// TwinCAT 3 PLC project TwinCAT_OpenFramework_Tasks
// Title: TwinCAT Open Framework Tasks
// Company: Oleksandr Tiutyk FOP
// Author: Oleksandr Tiutyk
// ProjectVersion: 1.0.13.0
// Description: TwinCAT.OpenFramework abstractions to run simple tasks
// ProgramVersion: 3.1.4026.28
// libraries:
//   [TwinCAT Open Framework Collections], * (Oleksandr Tiutyk FOP)
//   [TwinCAT Open Framework Core], * (Oleksandr Tiutyk FOP)
// project tree:
//   Internal/ CurrentNamespace.TcPOU, NamespaceExtractor.TcPOU
//   TaskQueue/ StandardTaskQueue.TcPOU (not stored), TaskQueue.TcPOU
//   Task/Enums/ TASK_PROCESSING_STATE.TcDUT (not stored), TASK_RUNNING_SUBSTATE.TcDUT, TASK_STATE.TcDUT (not stored), TASK_STOP_REASON.TcDUT (not stored)
//   Task/ ITask.TcIO, Task.TcPOU
//   Task/SubObjects/ TaskRunningSubstate.TcPOU (not stored), TaskState.TcPOU, TaskStopReason.TcPOU (not stored)
//   Version/ Global_Version.TcGVL
// (motion and I/O tree: see PLC project twincat_openframework_core)
// real-time tasks:
//   TASK PlcTask: cycle T#10ms, priority 20, ADS port 350
//   TASK TestTask: cycle T#10ms, priority 1, ADS port 351
//   TASK RunnerTestTask: cycle T#10ms, priority 2, ADS port 354
//   TASK HowToTask: cycle T#10ms, priority 22, ADS port 353
// variable links:

// ---- Task/Enums/TASK_RUNNING_SUBSTATE.TcDUT
(*
SPDX-FileCopyrightText: © 2026 Oleksandr Tiutyk <trofimich@gmail.com>
SPDX-License-Identifier: MIT
License: https://opensource.org/license/mit
*)

(*!
<summary>Identifies the active phase of a running task.</summary>
<description>
Acquisition, processing, stopping and release are diagnostic substates, not independent scheduling tasks.
Interpret them only while TASK_STATE is RUNNING.
</description>
*)
{attribute 'qualified_only'}
{attribute 'strict'}
{attribute 'to_string'}
TYPE TASK_RUNNING_SUBSTATE :
(
	//! <summary>Acquire the resource before ordinary work.</summary>
	RESOURCE_ACQUIRING := 0,
	//! <summary>Advance ordinary work unless cancellation is pending.</summary>
	PROCESSING,
	//! <summary>Advance the terminal resource-release attempt.</summary>
	RESOURCE_RELEASING,
	//! <summary>Finish active work for any stop reason before resource release.</summary>
	STOPPING
);
END_TYPE

// ---- Version/Global_Version.TcGVL
{attribute 'TcGenerated'}
{attribute 'no-analysis'}
{attribute 'linkalways'}
// This function has been automatically generated from the project information.
VAR_GLOBAL CONSTANT
	{attribute 'const_non_replaced'}
	stLibVersion_TwinCAT_Open_Framework_Tasks : ST_LibVersion := (iMajor := 1, iMinor := 0, iBuild := 13, iRevision := 0, nFlags := 0, sVersion := '1.0.13.0');
END_VAR

// ---- Task/ITask.TcIO
(*
SPDX-FileCopyrightText: © 2026 Oleksandr Tiutyk <trofimich@gmail.com>
SPDX-License-Identifier: MIT
License: https://opensource.org/license/mit
*)

(*!
<summary>Defines a reusable cooperative operation with optional resource acquisition and release.</summary>
<description>
One owner drives inherited Execute cyclically while RUNNING, including after an accepted Cancel, until
STOPPED. Avoid concurrent or recursive Execute on the same task. State, RunningSubstate and stop reasons are
borrowed live views for observation only; keep the task alive and do not modify referenced data. Copy result
values and messages before Reset or reuse. Boolean control results do not establish a general no-throw
guarantee for arbitrary implementations or diagnostic failures.
</description>
*)
INTERFACE ITask EXTENDS TOF_Core.IExecutable, TOF_Core.INamed

(*!
<summary>Requests cancellation before resource release begins.</summary>
<description>
Accepted only in RUNNING with no pending cancellation and before resource release. TRUE means accepted, not
completed; continue Execute until STOPPED. Accepted cancellation enters STOPPING, including from a previous
work result in that phase, and sets EXTERNAL_CANCEL. Repeated, releasing or non-running requests return FALSE
with refuseReason.
</description>
<param name="refuseReason">Reason for refusal; meaningful on FALSE.</param>
*)
METHOD Cancel : BOOL
VAR_OUTPUT
	refuseReason : TOF_Core.ERROR_MESSAGE;
END_VAR
END_METHOD

(*!
<summary>Provides the final lifecycle result for a stopped task.</summary>
<description>
Meaningful as a final result only in STOPPED. Release exceptions produce FAILURE without an automatic release
retry; STOPPED does not prove physical resource release. Best-effort errors handled inside the manager do not
by themselves change this result. Reset clears the message and restores the default reason. The view is
borrowed and read-only.
</description>
*)
{attribute 'monitoring' := 'call'}

PROPERTY FINAL FinalStopReason : REFERENCE TO TaskStopReason
GET
END_GET
END_PROPERTY

(*!
<summary>Provides the reason that initiated stopping.</summary>
<description>
Completion, internal abort, external cancellation or failure is preserved with its message during release; a
release exception affects FinalStopReason instead. The initial WORK_DONE value does not indicate completion.
Reset restores defaults. This is a borrowed read-only live view.
</description>
*)
{attribute 'monitoring' := 'call'}

PROPERTY FINAL OriginalStopReason : REFERENCE TO TaskStopReason
GET
END_GET
END_PROPERTY

(*!
<summary>Prepares a stopped task for reuse.</summary>
<description>
READY returns TRUE without callbacks or reinitialization. RUNNING refuses reset; cancel and keep calling
Execute until STOPPED first. In STOPPED, successful reset restores default stop reasons and clears their
messages. A refused reset does not guarantee rollback of callback effects.
</description>
<param name="refuseReason">Reason for refusal; meaningful on FALSE.</param>
*)
METHOD Reset : BOOL
VAR_OUTPUT
	refuseReason : TOF_Core.ERROR_MESSAGE;
END_VAR
END_METHOD

(*!
<summary>Provides the borrowed manager used by the task, or zero for none.</summary>
<description>
Keep the manager alive and stable throughout the run. The task issues StartAcquire or StartRelease once per
phase and advances Execute; external callers must not drive those operations concurrently. Pending acquisition
and active work must finish according to the concrete manager and task contracts before release.
ResourceManager and ResourceAcquired getters have no side effects and must not throw.
</description>
*)
{attribute 'monitoring' := 'call'}

PROPERTY ResourceManager : TOF_Core.IResourceManager
GET
END_GET
END_PROPERTY

(*!
<summary>Provides a live diagnostic view of the running phase.</summary>
<description>
Meaningful only while State.Running is TRUE. Observe acquisition, processing, stopping or release without
driving the resource manager directly. The view is borrowed and read-only.
</description>
*)
{attribute 'monitoring' := 'call'}

PROPERTY FINAL RunningSubstate : REFERENCE TO TaskRunningSubstate
GET
END_GET
END_PROPERTY

(*!
<summary>Starts a READY task's lifecycle.</summary>
<description>
TRUE means RUNNING, not completed. Continue Execute for work and cleanup. Ineligible state or refused
preparation returns FALSE with refuseReason. Refusal does not guarantee rollback of preparation already
performed.
</description>
<param name="refuseReason">Reason for refusal; meaningful on FALSE.</param>
*)
METHOD Start : BOOL
VAR_OUTPUT
	refuseReason : TOF_Core.ERROR_MESSAGE;
END_VAR
END_METHOD

(*!
<summary>Provides a live view of the task lifecycle.</summary>
<description>
READY precedes start, RUNNING includes acquisition, work, stopping and release, and STOPPED marks termination.
Assess the completed result through FinalStopReason. StateChanged is cleared at the start of Execute and set
on a lifecycle transition; its lifetime follows method calls, not necessarily one PLC cycle. The view is
borrowed and read-only.
</description>
*)
{attribute 'monitoring' := 'call'}

PROPERTY FINAL State : REFERENCE TO TaskState
GET
END_GET
END_PROPERTY

END_INTERFACE

// ---- Internal/CurrentNamespace.TcPOU
(*
SPDX-FileCopyrightText: © 2026 Oleksandr Tiutyk <trofimich@gmail.com>
SPDX-License-Identifier: MIT
License: https://opensource.org/license/mit
*)

(*!
<summary>Exposes this library's compiler-initialized namespace.</summary>
<description>
Internal metadata provider; no cyclic body call is needed. The returned namespace is borrowed read-only
storage.
</description>
*)

{attribute 'no_explicit_call' := 'do not call this POU directly'}
PROGRAM INTERNAL CurrentNamespace
VAR
	{attribute 'hide'} 
	_NamespaceExtractor : NamespaceExtractor;
END_VAR

(*!
<summary>Borrows the compiler-initialized library namespace.</summary>
<description>
Do not modify the referenced storage. Reading does not allocate or transfer ownership.
</description>
*)
{attribute 'monitoring' := 'call'}
PROPERTY Name : REFERENCE TO STRING
GET
Name REF= _NamespaceExtractor.CurrentNamespace;
END_GET
END_PROPERTY

END_PROGRAM

// ---- Internal/NamespaceExtractor.TcPOU
(*
SPDX-FileCopyrightText: © 2026 Oleksandr Tiutyk <trofimich@gmail.com>
SPDX-License-Identifier: MIT
License: https://opensource.org/license/mit
*)

(*!
<summary>Captures the current library namespace through init_namespace.</summary>
<description>
The compiler initializes CurrentNamespace. The empty body requires no execution; consumers treat the output as
read-only metadata.
</description>
*)

FUNCTION_BLOCK INTERNAL NamespaceExtractor
VAR_OUTPUT
	//! <summary>Compiler-supplied library namespace; read-only to consumers.</summary>
	{attribute 'init_namespace'} 
	CurrentNamespace : STRING;	
END_VAR

END_FUNCTION_BLOCK

// ---- TaskQueue/TaskQueue.TcPOU
(*
SPDX-FileCopyrightText: © 2026 Oleksandr Tiutyk <trofimich@gmail.com>
SPDX-License-Identifier: MIT
License: https://opensource.org/license/mit
*)

(*!
<summary>Executes borrowed child tasks sequentially in FIFO order.</summary>
<description>
One owner drives the queue and the lifecycles of its queued children. Children must be live, READY when
enqueued and unique in this queue; callers must not independently drive them while queued. Only one child is
active at a time. The dynamic list owns its storage but not child objects. Successful children are removed;
unsuccessful current and waiting entries remain until cleared or reset. Empty queues keep running unless
StopWhenNoPendingTasks is TRUE. All stop reasons advance the current child's cleanup without starting waiting
children. The base Task records a processing exception and enters STOPPING; OnStopping requests child
cancellation and waits for completion before parent release. An accepted external Cancel during that wait
retains the base Task cancellation result; the first failure is submitted to the log. No cleanup timeout is
imposed. Descendants overriding queue hooks must preserve the inherited queue operations.
</description>
*)

{attribute 'no_explicit_call' := 'do not call this function block directly'}
FUNCTION_BLOCK ABSTRACT TaskQueue EXTENDS Task
VAR
	{attribute 'hide'} 
	_SubTasks : TOF_Collections.List<0>(0);
	
	{attribute 'hide'} 
	_CurrentTask : ITask;
	
	{attribute 'hide'} 
	_StopWhenNoPendingTasks : BOOL;
END_VAR

(*!
<summary>Removes waiting entries without resetting or deleting child objects.</summary>
<description>
While RUNNING with a current task, retains that first entry and removes the rest. Otherwise clears all entries
and the current reference. Does not request cancellation. A stopped unsuccessful current task is removed when
clearing outside RUNNING.
</description>
*)
METHOD FINAL ClearWaitingTasks
VAR
	i : DINT;
END_VAR
IF NOT State.Running OR_ELSE _CurrentTask = 0 THEN
	_SubTasks.Clear();
	_CurrentTask := 0;
ELSE	
	FOR i := _SubTasks.Length - 1 TO 1 BY -1 DO
		_SubTasks.RemoveAt(index := i);
	END_FOR
END_IF
END_METHOD

(*!
<summary>Appends a prepared borrowed task to the FIFO.</summary>
<description>
Null raises ArgumentNotSpecifiedException. READY and uniqueness are caller preconditions, not checked here.
Keep the child alive and do not start, execute, cancel or reset it independently while queued. Removal
transfers no ownership and does not reset or delete it. No queue-state guard is applied; Reset from STOPPED
clears entries, so prepare the queue before filling it for reuse. Storage growth can raise terminal allocation
failure.
</description>
<param name="task">Live READY child whose lifecycle is delegated to the queue until removal.</param>
*)
METHOD PROTECTED FINAL EnqueueTask
VAR_INPUT
	task : ITask;
END_VAR
VAR
	
	taskAsGeneric : TOF_Core.GENERIC_VALUE;
END_VAR
IF task = 0 THEN
	TOF_Core.Exceptions.ThrowArgumentNotSpecified(
		sourceNamespaceName := NamespaceName,
		sourceClassName := ClassName,
		sourcePOUName := __POUNAME(),
		sourcePosition := __POSITION(),
		argumentName := 'task'
	);
END_IF

taskAsGeneric := TOF_Core.GenericValueFactory.FromParts(
		genericTypeClass := TOF_Core.GENERIC_TYPE_CLASS.OBJECT,
		address := task.SelfAddress,
		size := task.SelfSize,
		memoryManagementBehavior := TOF_Core.GENERIC_MEMORY_MANAGEMENT_BEHAVIOR.STORE_ORIGINAL_REFERENCE_AND_NOT_OWNS_MEMORY
	);

_SubTasks.AppendGeneric(value := taskAsGeneric);
END_METHOD

(*!
<summary>Resolves one stored entry to its task interface.</summary>
<description>
Requires a valid zero-based index and a live borrowed child. List access rejects an invalid index; failure to
query ITask raises StandardException. Does not clone or transfer ownership.
</description>
<param name="index">Index within the queue's current list.</param>
*)
METHOD PRIVATE getTaskByIndex : ITask
VAR_INPUT
	index : DINT;
END_VAR
VAR
	taskInterface : TOF_Core.IObject;
	
END_VAR
taskInterface := _SubTasks.Get(index := index).AsIObject();

IF NOT __QUERYINTERFACE(taskInterface, getTaskByIndex) THEN
	TOF_Core.Exceptions.ThrowStandard(
		sourceNamespaceName := NamespaceName,
		sourceClassName := ClassName,
		sourcePOUName := __POUNAME(),
		sourcePosition := __POSITION(),
		message := "Can't convert task from _Tasks collection to ITask type"
	);
END_IF
END_METHOD

(*!
<summary>Cancels and advances the current child before any parent termination.</summary>
<description>
Called by the common STOPPING phase after any result or exception. Never starts waiting children. Requests
Cancel while the child is RUNNING, then advances it once. A Cancel exception is contained so Execute still
gets a chance to progress; readiness remains FALSE for that call. Execute exceptions reach the base stopping
handler, which retains the original result and retries. Refusal of Cancel does not imply completion. No child
is removed or reset here. Additional descendant cleanup must combine readiness with this result.
</description>
<param name="readyToRelease">TRUE when no child is RUNNING and this stopping step completed normally.</param>
*)
METHOD PROTECTED OnStopping
VAR_OUTPUT
	readyToRelease : BOOL;
END_VAR
VAR
	cancelCallFailed : BOOL;
END_VAR
IF _CurrentTask <> 0 AND_THEN _CurrentTask.State.Running THEN
	__TRY
		_CurrentTask.Cancel();
	__CATCH
		// Advance the child even if its cancellation request was interrupted.
		cancelCallFailed := TRUE;
	__ENDTRY

	_CurrentTask.Execute();
END_IF

readyToRelease := NOT cancelCallFailed
	AND_THEN (_CurrentTask = 0 OR_ELSE NOT _CurrentTask.State.Running);
END_METHOD

(*!
<summary>Forwards an accepted queue cancellation to its running child.</summary>
<description>
Called once by the task's Cancel path. Does not wait or inspect the child's refusal message; a child already
stopping can refuse another cancellation request. OnStopping advances completion. Preserve forwarding when
overriding this hook.
</description>
*)
METHOD PROTECTED OnCancelRequest
IF _CurrentTask <> 0 AND_THEN _CurrentTask.State.Running THEN
	_CurrentTask.Cancel();
END_IF
END_METHOD

(*!
<summary>Clears a stopped queue for reuse.</summary>
<description>
Releases list storage and drops current and waiting references without resetting or deleting children. Their
owner prepares them before re-enqueueing. Base Reset clears stop diagnostics. READY Reset does not invoke this
hook; use ClearWaitingTasks to empty a READY queue. Descendants must preserve this step.
</description>
*)
METHOD PROTECTED OnReset
_SubTasks.Clear();
_CurrentTask := 0;
END_METHOD

(*!
<summary>Starts or advances at most one current child per processing call.</summary>
<description>
An existing current child receives one Execute. Otherwise the first waiting child is selected and started;
newly started work is advanced by a later call. Start refusal or an unexpected READY current yields ERROR. A
successful stopped child is removed; other results are mapped from FinalStopReason and its message. An empty
queue yields DONE only when StopWhenNoPendingTasks is TRUE. Removing the last successful child leaves BUSY
until the next call. Exceptions propagate to the base Task failure handler, which records and logs diagnostics
and enters STOPPING. OnStopping waits for child cleanup before parent release.
</description>
<param name="processingState">Queue progress; defaults to BUSY while waiting or advancing a child.</param>
<param name="stopReasonMessage">Receives child refusal or unsuccessful completion diagnostics.</param>
*)
METHOD PROTECTED OnRunning
VAR_OUTPUT
	processingState : TASK_PROCESSING_STATE;
END_VAR
VAR_IN_OUT
	stopReasonMessage : TOF_Core.ERROR_MESSAGE;
END_VAR
IF _CurrentTask <> 0 THEN
	_CurrentTask.Execute();
ELSIF _SubTasks.Length > TOF_Core.SignedInt32.ZERO THEN
	_CurrentTask := getTaskByIndex(index := 0);

	IF NOT _CurrentTask.Start(refuseReason => stopReasonMessage) THEN
		processingState := TASK_PROCESSING_STATE.ERROR;
		RETURN;
	END_IF
ELSIF _StopWhenNoPendingTasks THEN
	processingState := TASK_PROCESSING_STATE.DONE;
END_IF

IF _CurrentTask <> 0 THEN
	CASE _CurrentTask.State.Value OF
		TASK_STATE.READY:
			processingState := TASK_PROCESSING_STATE.ERROR;
			stopReasonMessage := "Current task returned to READY before completion";

		TASK_STATE.STOPPED:
			IF _CurrentTask.FinalStopReason.WorkDone THEN
				removeCurrentTask();
			ELSE
				processingState := GetProcessingStateByStopReason(taskStopReason := _CurrentTask.FinalStopReason.Value);
				stopReasonMessage := _CurrentTask.FinalStopReason.Message;
			END_IF
	END_CASE
END_IF
END_METHOD

(*!
<summary>Reports the number of entries still retained by the queue.</summary>
<description>
Includes the current task and waiting children, including a failed or cancelled current retained after
stopping. Zero does not by itself mean the queue has reached STOPPED.
</description>
*)
{attribute 'monitoring' := 'call'}
PROPERTY FINAL PendingTaskCount : DINT
GET
PendingTaskCount := _SubTasks.Length;
END_GET
END_PROPERTY

(*!
<summary>Removes the first queue entry and clears the current reference.</summary>
<description>
Used after successful child completion. Compacts remaining list entries without resetting or deleting the
child; the caller retains its object and may inspect its stopped result. Does not start the next child.
</description>
*)
METHOD PRIVATE removeCurrentTask
IF _SubTasks.Length > 0 THEN
	_SubTasks.RemoveAt(index := 0);
END_IF

_CurrentTask := 0;
END_METHOD

(*!
<summary>Controls whether an empty running queue completes.</summary>
<description>
Defaults to FALSE, allowing Execute to wait for later enqueueing. TRUE makes OnRunning report DONE when it
finds no current or waiting child. May be changed between owner calls; setting it does not itself execute or
stop the queue.
</description>
*)
{attribute 'monitoring' := 'call'}
PROPERTY FINAL StopWhenNoPendingTasks : BOOL
GET
StopWhenNoPendingTasks := _StopWhenNoPendingTasks;
END_GET
SET
_StopWhenNoPendingTasks := StopWhenNoPendingTasks;
END_SET
END_PROPERTY

END_FUNCTION_BLOCK

// ---- Task/Task.TcPOU
(*
SPDX-FileCopyrightText: © 2026 Oleksandr Tiutyk <trofimich@gmail.com>
SPDX-License-Identifier: MIT
License: https://opensource.org/license/mit
*)

(*!
<summary>Runs a reusable cooperative operation through acquisition, processing, stopping and release.</summary>
<description>
One owner drives the task through Start, cyclic Execute and Reset; no worker thread or PLC scheduler task is
created. Keep callbacks short and avoid concurrent or recursive Execute. The resource manager is borrowed and
must remain live and stable during a run. All stop reasons wait through OnStopping before release. Normal work
completion advances stopping in the same Execute, without waiting or repeating work. No callback may
recursively drive this task, except Reset in OnAfterStop. Ordinary work and resource exceptions are converted
into stop diagnostics where handled. If obtaining their messages fails, phase-specific fallback text preserves
the intended failure transition; preparation and reset use the same fallback policy for refusal. The first
stopping exception is submitted to the log; later stopping exceptions retry without repeated log attempts.
This is not a universal no-throw boundary. The caller still provides exception cleanup and terminal
allocation-failure checks at its PLC task boundary. DiagnosticLogger optionally selects an independent
diagnostic channel; zero preserves LogManager routing. Configure it before Start and keep it stable until
STOPPED, including Reset diagnostics, with no concurrent access.
</description>
*)

{attribute 'no_explicit_call' := 'do not call this function block directly'}
FUNCTION_BLOCK ABSTRACT Task EXTENDS TOF_Core.Object IMPLEMENTS ITask
VAR
	{attribute 'hide'} 
	_Name : WSTRING;

	//! <summary>Optional borrowed destination for this task's internal diagnostics.</summary>
	_DiagnosticLogger : TOF_Core.ILogger;
	
	{attribute 'hide'} 
	_State : TASK_STATE;	
	{attribute 'hide'} 
	_StateChanged : BOOL;	
	{attribute 'hide'} 
	_RunningSubstate : TASK_RUNNING_SUBSTATE;
	{attribute 'hide'} 
	_ResourceOperationStarted : BOOL;
	//! <summary>Tracks whether a stopping exception has been submitted to the log in this run.</summary>
	{attribute 'hide'}
	_StoppingExceptionReportAttempted : BOOL;

	{attribute 'hide'} 
	_OriginalStopReason : TASK_STOP_REASON;
	{attribute 'hide'} 
	_TemporaryErrorMessage : TOF_Core.ERROR_MESSAGE;	
	{attribute 'hide'} 
	_OriginalStopReasonMessage : TOF_Core.ERROR_MESSAGE;
	{attribute 'hide'} 
	_OriginalStopReasonObject : TaskStopReason(_OriginalStopReason, _OriginalStopReasonMessage);
	
	{attribute 'hide'} 
	_FinalStopReason : TASK_STOP_REASON;	
	{attribute 'hide'} 
	_FinalStopReasonMessage : TOF_Core.ERROR_MESSAGE;
	{attribute 'hide'} 
	_FinalStopReasonObject : TaskStopReason(_FinalStopReason, _FinalStopReasonMessage);
	
	{attribute 'hide'} 
	_StateObject : TaskState(_State, _StateChanged);
	{attribute 'hide'} 
	_RunningSubstateObject : TaskRunningSubstate(_RunningSubstate);
END_VAR

(*!
<summary>Requests cooperative cancellation of a running task.</summary>
<description>
Accepted only while RUNNING, with no pending cancellation and before RESOURCE_RELEASING. Records
EXTERNAL_CANCEL as the original reason and enters STOPPING before invoking OnCancelRequest once. A first
Cancel during STOPPING replaces the original result with EXTERNAL_CANCEL. TRUE means accepted, not completed;
continue Execute until STOPPED. Repeated or ineligible requests return FALSE with refuseReason. Callback
exceptions are logged without withdrawing the request.
</description>
<param name="refuseReason">Reason for refusal; meaningful when the method returns FALSE.</param>
*)
METHOD FINAL Cancel : BOOL
VAR_OUTPUT
	refuseReason : TOF_Core.ERROR_MESSAGE;
END_VAR
IF _State <> TASK_STATE.RUNNING THEN
	refuseReason := TOF_Core.WideStrings.Concat255(
		"Expected state is '",
		TO_WSTRING(TASK_STATE.RUNNING),
		"' but current state is '",
		TO_WSTRING(_State),
		"'"
	);
	RETURN;
END_IF

IF _OriginalStopReason = TASK_STOP_REASON.EXTERNAL_CANCEL
	OR_ELSE _RunningSubstate = TASK_RUNNING_SUBSTATE.RESOURCE_RELEASING
THEN
	refuseReason := "Cancellation already requested or resource release has begun";
	RETURN;
END_IF

_OriginalStopReason := TASK_STOP_REASON.EXTERNAL_CANCEL;
_OriginalStopReasonMessage := "Cancelled by external logic";

setRunningSubstate(runningSubState := TASK_RUNNING_SUBSTATE.STOPPING);

safeCallOnCancelRequest();

Cancel := TRUE;
END_METHOD

(*!
<summary>Advances the running task and clears its transition indicator.</summary>
<description>
Clears State.StateChanged on every call, including READY and STOPPED calls. While RUNNING, advances
acquisition, work or release without a blocking wait. A normal terminal work result also advances stopping
once in the same call. A caught acquire/process exception defers stopping until the next Execute. Readiness
selects release for a later Execute, or stops immediately without a resource. The owner determines call
frequency and must keep calling during cleanup. No automatic scheduling or general callback reentrancy
protection is provided.
</description>
*)
METHOD FINAL Execute
_StateChanged := FALSE;

IF _State = TASK_STATE.RUNNING THEN
	handleRunning();
END_IF
END_METHOD

(*!
<summary>Stores an explicit diagnostic name or constructs the default name during initialization.</summary>
<description>
Copies a nonempty name into task-owned storage. For an empty name, stores Object.GetDefaultName using ClassName
and the instance address. Overridden ClassName must be ready during base initialization, use initialized static
storage without derived instance dependencies, and neither raise exceptions nor recursively read Name.
Does not start work or acquire resources. Start and Reset preserve the name. Skipped during online change copy
code so the copied name remains unchanged.
</description>
<param name="name">Diagnostic name to copy, or empty to request the default name.</param>
*)
METHOD FB_init : BOOL
VAR_INPUT	
	bInitRetains : BOOL; // TRUE: the retain variables are initialized (reset warm / reset cold)
	bInCopyCode : BOOL;  // TRUE: the instance will be copied to the copy code afterward (online change)
	name : WSTRING;
END_VAR
IF NOT bInCopyCode THEN
	IF name <> TOF_Core.WideStrings.Empty THEN
		_Name := name;
	ELSE
		_Name := GetDefaultName();
	END_IF
END_IF
END_METHOD

(*!
<summary>Restores internal view bindings after an online change.</summary>
<description>
Implicitly called by the runtime after instance copy code completes. Rebinds internal view objects to
the current instance fields to repair any references relocated during the online change.
</description>
*)
METHOD FB_reinit : BOOL
_OriginalStopReasonObject.Rebind(
	stopReason := _OriginalStopReason,
	stopReasonMessage := ADR(_OriginalStopReasonMessage)
);
_FinalStopReasonObject.Rebind(
	stopReason := _FinalStopReason,
	stopReasonMessage := ADR(_FinalStopReasonMessage)
);
_StateObject.Rebind(
	taskState := _State,
	taskStateChanged := _StateChanged
);
_RunningSubstateObject.Rebind(
	taskRunningSubstate := _RunningSubstate
);

FB_reinit := TRUE;
END_METHOD

(*!
<summary>Final termination result; meaningful as a final result only in STOPPED.</summary>
<description>
STOPPED means execution has ended, not that physical resource release succeeded. Resource-release exceptions
produce FAILURE without an automatic release retry. Best-effort errors handled and logged by the resource
manager do not by themselves change this result. Reset restores the default reason and clears the message.
This is a live view.
</description>
*)

{attribute 'monitoring' := 'call'}
PROPERTY FINAL FinalStopReason : REFERENCE TO TaskStopReason
GET
FinalStopReason REF= _FinalStopReasonObject;
END_GET
END_PROPERTY

(*!
<summary>Maps a completed task's stop reason to a processing result.</summary>
<description>
WORK_DONE maps to DONE, INTERNAL_ABORT and EXTERNAL_CANCEL to ABORTED, and FAILURE to ERROR. Call with a
defined TASK_STOP_REASON after completion. No state is modified; an unrecognized value is not rejected and
leaves the default BUSY result.
</description>
<param name="taskStopReason">Completed task result to translate.</param>
*)
METHOD PROTECTED GetProcessingStateByStopReason : TASK_PROCESSING_STATE
VAR_INPUT
	taskStopReason : TASK_STOP_REASON;
END_VAR
CASE taskStopReason OF
	TASK_STOP_REASON.WORK_DONE:
		GetProcessingStateByStopReason := TASK_PROCESSING_STATE.DONE;
	
    TASK_STOP_REASON.INTERNAL_ABORT, TASK_STOP_REASON.EXTERNAL_CANCEL:
		GetProcessingStateByStopReason := TASK_PROCESSING_STATE.ABORTED;
	
    TASK_STOP_REASON.FAILURE:
		GetProcessingStateByStopReason := TASK_PROCESSING_STATE.ERROR;
END_CASE
END_METHOD

(*!
<summary>Maps a terminal processing result to the reason for stopping.</summary>
<description>
DONE maps to WORK_DONE, ABORTED to INTERNAL_ABORT, and ERROR to FAILURE. BUSY and unrecognized values raise
ArgumentOutOfRangeException. Does not modify task state.
</description>
<param name="taskpPocessingState">Terminal result from OnRunning.</param>
*)
METHOD PROTECTED GetStopReasonByProcessingState : TASK_STOP_REASON
VAR_INPUT
	taskpPocessingState : TASK_PROCESSING_STATE;
END_VAR
VAR
	
	taskRunningResultName : STRING(16);
END_VAR
CASE taskpPocessingState OF
	TASK_PROCESSING_STATE.DONE:
		GetStopReasonByProcessingState := TASK_STOP_REASON.WORK_DONE;
	
    TASK_PROCESSING_STATE.ABORTED:
		GetStopReasonByProcessingState := TASK_STOP_REASON.INTERNAL_ABORT;
		
    TASK_PROCESSING_STATE.ERROR:
		GetStopReasonByProcessingState := TASK_STOP_REASON.FAILURE;
	
	ELSE
		taskRunningResultName := TO_STRING(taskpPocessingState);
		TOF_Core.Exceptions.ThrowArgumentOutOfRange(
			sourceNamespaceName := NamespaceName,
			sourceClassName := ClassName,
			sourcePOUName := __POUNAME(),
			sourcePosition := __POSITION(),
			argumentName := 'taskpPocessingState',
			argumentValue := taskRunningResultName
		);
END_CASE
END_METHOD

(*!
<summary>Advances work and permits immediate stopping after a normal terminal result.</summary>
<description>
Every terminal work result and acquire/process exception enters STOPPING. Normal results call OnStopping once
immediately; exceptions leave its first call for the next Execute to avoid advancing a failed child twice in
one call. OnStopping must complete before release or STOPPED; its exceptions keep STOPPING without replacing
the original reason. The first stopping exception is submitted to the log; later ones retry without another
log attempt. Release exceptions terminate the attempt with final FAILURE and no retry. A caught exception uses
named, phase-specific fallback text if its message is empty or formatting fails; fixed phase text remains if
fallback formatting also fails. Terminal allocation failure remains latched for the owner's fatal boundary.
Callbacks must not recursively drive this task; OnAfterStop may Reset after finalization.
</description>
*)
METHOD PRIVATE handleRunning
VAR
	readyToRelease : BOOL;
	taskProcessingState : TASK_PROCESSING_STATE;
	exceptionCode : __SYSTEM.ExceptionCode;
	exception : TOF_Core.IException;
	phaseFailureMessage : WSTRING(40);
END_VAR
__TRY

	CASE _RunningSubstate OF
		TASK_RUNNING_SUBSTATE.RESOURCE_ACQUIRING:

			IF NOT _ResourceOperationStarted THEN
				_ResourceOperationStarted := TRUE;

				ResourceManager.StartAcquire();
			END_IF

			ResourceManager.Execute();

			IF ResourceManager.ResourceAcquired THEN
				setRunningSubstate(runningSubState := TASK_RUNNING_SUBSTATE.PROCESSING);
			END_IF

		TASK_RUNNING_SUBSTATE.PROCESSING:
			OnRunning(processingState => taskProcessingState, stopReasonMessage := _OriginalStopReasonMessage);

			IF taskProcessingState <> TASK_PROCESSING_STATE.BUSY THEN
				_OriginalStopReason := GetStopReasonByProcessingState(taskpPocessingState := taskProcessingState);
				setRunningSubstate(runningSubState := TASK_RUNNING_SUBSTATE.STOPPING);
			END_IF

		TASK_RUNNING_SUBSTATE.RESOURCE_RELEASING:

			IF NOT _ResourceOperationStarted THEN
				_ResourceOperationStarted := TRUE;

				ResourceManager.StartRelease();
			END_IF

			ResourceManager.Execute();

			IF NOT ResourceManager.ResourceAcquired THEN
				setStoppedState(finalStopReason := _OriginalStopReason, finalStopReasonMessage := _OriginalStopReasonMessage);
				safeCallOnAfterStop();
			END_IF

	END_CASE

	IF _State = TASK_STATE.RUNNING AND_THEN _RunningSubstate = TASK_RUNNING_SUBSTATE.STOPPING THEN
		OnStopping(readyToRelease => readyToRelease);

		IF readyToRelease THEN

			IF ReleaseResourceRequired THEN
				setRunningSubstate(runningSubState := TASK_RUNNING_SUBSTATE.RESOURCE_RELEASING);
			ELSE
				setStoppedState(finalStopReason := _OriginalStopReason, finalStopReasonMessage := _OriginalStopReasonMessage);
				safeCallOnAfterStop();
			END_IF

		END_IF

	END_IF

__CATCH(exceptionCode)
	IF _RunningSubstate = TASK_RUNNING_SUBSTATE.STOPPING THEN

		IF _StoppingExceptionReportAttempted THEN
			// Continue the interrupted hook on a later Execute without repeated logging.
			RETURN;
		END_IF

		_StoppingExceptionReportAttempted := TRUE;
	END_IF

	CASE _RunningSubstate OF
		TASK_RUNNING_SUBSTATE.RESOURCE_ACQUIRING:
			phaseFailureMessage := "resource acquisition failed";

		TASK_RUNNING_SUBSTATE.PROCESSING:
			phaseFailureMessage := "processing failed";

		TASK_RUNNING_SUBSTATE.STOPPING:
			phaseFailureMessage := "stopping failed";

		TASK_RUNNING_SUBSTATE.RESOURCE_RELEASING:
			phaseFailureMessage := "release failed";
	END_CASE

	_TemporaryErrorMessage := phaseFailureMessage;

	__TRY
		_TemporaryErrorMessage := TOF_Core.WideStrings.Concat255("Task '", Name, "' ", phaseFailureMessage);
		exception := TOF_Core.ExceptionManager.GetLastException(
			exceptionCode := exceptionCode,
			catchPointNamespaceName := NamespaceName,
			catchPointPOUName := __POUNAME(),
			catchPointPosition := __POSITION()
		);
		_TemporaryErrorMessage := exception.GetMessage();

		IF _TemporaryErrorMessage = TOF_Core.WideStrings.Empty THEN
			_TemporaryErrorMessage := phaseFailureMessage;
			_TemporaryErrorMessage := TOF_Core.WideStrings.Concat255("Task '", Name, "' ", phaseFailureMessage);
		END_IF

	__CATCH
		// Keep the named or fixed phase fallback and any terminal allocation-failure latch.
	__ENDTRY

	TryLogDiagnosticMessage(
		message := _TemporaryErrorMessage,
		category := TOF_Core.LOG_CATEGORY.ERROR,
		topic1 := "Task",
		topic2 := "Execute"
	);

	CASE _RunningSubstate OF
		TASK_RUNNING_SUBSTATE.RESOURCE_RELEASING:
			setStoppedState(finalStopReason := TASK_STOP_REASON.FAILURE, finalStopReasonMessage := _TemporaryErrorMessage);
			safeCallOnAfterStop();

		TASK_RUNNING_SUBSTATE.STOPPING:
			// Retry stopping later; never release after an interrupted hook.
			RETURN;

		ELSE
			_OriginalStopReason := TASK_STOP_REASON.FAILURE;
			_OriginalStopReasonMessage := _TemporaryErrorMessage;

			setRunningSubstate(runningSubState := TASK_RUNNING_SUBSTATE.STOPPING);
	END_CASE

__ENDTRY
END_METHOD

(*!
<summary>Provides the task's diagnostic name.</summary>
<description>
FB_init stores the supplied name or constructs the default from ClassName and the instance address. Reading
only borrows the stored buffer; it does not initialize or recompute metadata, start work or synchronize callers.
Start and Reset preserve the name and its storage. The returned reference remains valid while the task lives;
do not write through it. The name is diagnostic text, not a persistent identifier; later ClassName changes or
instance relocation do not rename the task.
</description>
*)

{attribute 'monitoring' := 'call'}
PROPERTY FINAL Name : REFERENCE TO WSTRING
GET
Name REF= _Name;
END_GET
END_PROPERTY

(*!
<summary>Notifies descendants after final termination has been recorded.</summary>
<description>
Called after transition to STOPPED and assignment of FinalStopReason, following the release attempt when
required. Use for short notifications or bookkeeping for any stop reason. Callback exceptions are logged and
do not replace the recorded result. Reset from this hook can change the visible state and clear results before
Execute returns; it does not schedule another run. General recursive lifecycle control is not guaranteed.
</description>
*)
METHOD PROTECTED OnAfterStop
END_METHOD

(*!
<summary>Prepares a READY task synchronously before starting.</summary>
<description>
Called by Start before RUNNING and resource acquisition. Validate or prepare one run without waiting in a
loop. A callback exception refuses Start and supplies refuseReason, using fixed fallback text if obtaining the
exception message fails. Preparation already performed is not rolled back. The base does nothing.
</description>
*)
METHOD PROTECTED OnBeforeStart
END_METHOD

(*!
<summary>Initiates an accepted cancellation once.</summary>
<description>
Called synchronously by Cancel after the original stop reason is set to EXTERNAL_CANCEL. Not called for
refused or repeated requests. Initiate only short cancellation actions; Execute and OnStopping advance
completion. Callback exceptions are logged without withdrawing the request. The base implementation does
nothing.
</description>
*)
METHOD PROTECTED OnCancelRequest
END_METHOD

(*!
<summary>Resets descendant state before returning a stopped task to READY.</summary>
<description>
Called synchronously by Reset only in STOPPED, before base stop reasons and cancellation state are cleared.
READY Reset does not call this hook. A callback exception refuses Reset, using fixed fallback text if
obtaining the exception message fails; changes already made are not rolled back. The base implementation does
nothing. Descendants must preserve any reset work required by their immediate base class.
</description>
*)
METHOD PROTECTED OnReset
END_METHOD

(*!
<summary>Advances one step of the operation after resource acquisition.</summary>
<description>
Called only in PROCESSING. Return BUSY to continue, DONE to complete, ABORTED for internal abort or ERROR for
failure. A normal terminal result enters STOPPING and calls OnStopping once in the same Execute. The stop
message is the task's live per-run buffer and is not cleared before every callback. Exceptions enter the
task's failure and cleanup path; completed side effects are not rolled back. Keep execution bounded and do not
block waiting for an asynchronous result.
</description>
<param name="processingState">Result of this processing step; the default value is BUSY.</param>
<param name="stopReasonMessage">Optional diagnostic message retained for termination; not an owned buffer.</param>
*)
METHOD PROTECTED ABSTRACT OnRunning
VAR_OUTPUT
	processingState : TASK_PROCESSING_STATE;
END_VAR
VAR_IN_OUT
	stopReasonMessage : TOF_Core.ERROR_MESSAGE;
END_VAR
END_METHOD

(*!
<summary>Finishes active work before resource release for every stop reason.</summary>
<description>
Called in STOPPING after success, internal abort, failure or external cancellation. A normal terminal work
result invokes this hook in the same Execute; a caught work/acquire exception defers it to the next call.
Ordinary OnRunning and acquisition no longer execute. Set readyToRelease on every call; FALSE requires another
Execute. Finish pending I/O and acquisition without starting new work. TRUE permits release on the next
Execute, or immediate STOPPED when no resource is acquired. The base returns TRUE. An exception keeps STOPPING
and retries on a later Execute without changing the original result. Only the first stopping exception is
submitted to the log in a run; later ones are suppressed. Partial hook effects are not rolled back. Make
interrupted progress resumable. No timeout or physical abort is implied. Descendants must preserve inherited
stopping work and combine readiness.
</description>
<param name="readyToRelease">TRUE when active work no longer prevents release or termination.</param>
*)
METHOD PROTECTED OnStopping
VAR_OUTPUT
	readyToRelease : BOOL;
END_VAR
readyToRelease := TRUE;
END_METHOD

(*!
<summary>Reason recorded for stopping: completion, internal abort, cancellation or failure.</summary>
<description>
Established when stopping begins and preserved during resource release, along with its message. Release
exceptions affect FinalStopReason and its message. The initial WORK_DONE value does not indicate completed
work. Reset restores the default reason and clears the message. This is a live view.
</description>
*)

{attribute 'monitoring' := 'call'}
PROPERTY FINAL OriginalStopReason : REFERENCE TO TaskStopReason
GET
OriginalStopReason REF= _OriginalStopReasonObject;
END_GET
END_PROPERTY

(*!
<summary>Reports whether the current manager has an acquired resource.</summary>
<description>
TRUE only for a nonzero ResourceManager reporting ResourceAcquired. Does not initiate cleanup or determine
whether acquisition is still pending. Both getters must be non-throwing and free of side effects.
</description>
*)
{attribute 'monitoring' := 'call'}
PROPERTY PROTECTED FINAL ReleaseResourceRequired : BOOL
GET
VAR
	currentResourceManager : TOF_Core.IResourceManager;
END_VAR
currentResourceManager := ResourceManager;

ReleaseResourceRequired := currentResourceManager <> 0 AND_THEN currentResourceManager.ResourceAcquired;
END_GET
END_PROPERTY

(*!
<summary>Prepares a stopped task for reuse.</summary>
<description>
READY returns TRUE without callbacks or clearing state. RUNNING returns FALSE; cancel and drive Execute to
STOPPED first. In STOPPED, OnReset must succeed before base state returns to READY and stop diagnostics are
cleared. Partial callback effects are not rolled back on refusal. Failure to obtain a callback exception's
message uses fixed refusal text; terminal allocation failure still requires the caller's task-boundary check.
</description>
<param name="refuseReason">Reason for refusal; meaningful when the method returns FALSE.</param>
*)
METHOD FINAL Reset : BOOL
VAR_OUTPUT
	refuseReason : TOF_Core.ERROR_MESSAGE;
END_VAR
IF _State = TASK_STATE.READY THEN
	Reset := TRUE;
	RETURN;
END_IF

IF _State <> TASK_STATE.STOPPED THEN
	refuseReason := TOF_Core.WideStrings.Concat255(
		"Expected state is '",
		TO_WSTRING(TASK_STATE.READY),
		" or ",
		TO_WSTRING(TASK_STATE.STOPPED),
		"' but current state is '",
		TO_WSTRING(_State),
		"'"
	);
	RETURN;
END_IF
	
IF safeCallOnReset(refuseReason := refuseReason) THEN
	setIdleState();

	Reset := TRUE;
END_IF
END_METHOD

(*!
<summary>Provides the borrowed manager used for resource acquisition and release.</summary>
<description>
The base returns zero. Keep a nonzero manager alive and stable throughout the run; only the task drives its
StartAcquire, StartRelease and Execute methods. Start skips acquisition when already acquired, but normal
stopping still releases an acquired resource. During OnStopping, descendants must complete pending acquisition
as required by the manager before permitting release for any stop reason. Release exceptions terminate the
attempt with final FAILURE and no automatic retry. ResourceManager and ResourceAcquired getters must not throw
or have side effects.
</description>
*)

{attribute 'monitoring' := 'call'}
PROPERTY ResourceManager : TOF_Core.IResourceManager
GET
END_GET
END_PROPERTY

(*!
<summary>Provides a live read-only view of the current execution phase.</summary>
<description>
Meaningful only while State.Running is TRUE. The view borrows this task's fields and must not outlive it.
Observing a phase does not authorize external callers to drive the resource manager.
</description>
*)
{attribute 'monitoring' := 'call'}
PROPERTY FINAL RunningSubstate : REFERENCE TO TaskRunningSubstate
GET
RunningSubstate REF= _RunningSubstateObject;
END_GET
END_PROPERTY

(*!
<summary>Invokes the termination hook and attempts to log a callback exception.</summary>
<description>
Does not change the final result to reflect callback failure. Logging is best effort; a callback can already
have changed observable task state. Exception transport requires cyclic task context.
</description>
*)
METHOD PRIVATE safeCallOnAfterStop
VAR
	exceptionCode : __SYSTEM.ExceptionCode;
	exception : TOF_Core.IException;
END_VAR
__TRY
	OnAfterStop();
__CATCH(exceptionCode)
	exception := TOF_Core.ExceptionManager.GetLastException(
		exceptionCode := exceptionCode,
		catchPointNamespaceName := NamespaceName,
		catchPointPOUName := __POUNAME(),
		catchPointPosition := __POSITION()
	);

	TryLogDiagnosticException(
		exception := exception,
		severity := TOF_Core.ERROR_SEVERITY.ERROR,
		topic1 := TO_WSTRING(ClassName),
		topic2 := TO_WSTRING(__POUNAME())
	);
__ENDTRY
END_METHOD

(*!
<summary>Invokes start preparation and converts a callback exception to refusal.</summary>
<description>
Returns TRUE when OnBeforeStart returns normally. On exception, copies its formatted message to refuseReason
and leaves FALSE. If obtaining the message raises, retains fixed refusal text. Does not roll back callback
effects or clear terminal allocation failure; the caller's fatal boundary remains required.
</description>
<param name="refuseReason">Receives formatted diagnostics when preparation throws.</param>
*)
METHOD PRIVATE safeCallOnBeforeStart : BOOL
VAR_IN_OUT
	refuseReason : TOF_Core.ERROR_MESSAGE;
END_VAR
VAR
	exceptionCode : __SYSTEM.ExceptionCode;	
	exception : TOF_Core.IException;
END_VAR
__TRY
	OnBeforeStart();
	
	safeCallOnBeforeStart := TRUE;
__CATCH(exceptionCode)
	refuseReason := "Task start preparation failed";

	__TRY
		exception := TOF_Core.ExceptionManager.GetLastException(
			exceptionCode := exceptionCode,
			catchPointNamespaceName := NamespaceName,
			catchPointPOUName := __POUNAME(),
			catchPointPosition := __POSITION()
		);
		refuseReason := exception.GetMessage();
	__CATCH
		// Keep the fallback text and any terminal allocation-failure latch.
	__ENDTRY
__ENDTRY
END_METHOD

(*!
<summary>Invokes the cancellation notification and attempts to log a callback exception.</summary>
<description>
The cancellation request has already been accepted; callback failure does not undo the recorded reason.
Exception transport requires cyclic task context.
</description>
*)
METHOD PRIVATE safeCallOnCancelRequest
VAR
	exceptionCode : __SYSTEM.ExceptionCode;
	exception : TOF_Core.IException;
END_VAR
__TRY
	OnCancelRequest();
__CATCH(exceptionCode)
	exception := TOF_Core.ExceptionManager.GetLastException(
		exceptionCode := exceptionCode,
		catchPointNamespaceName := NamespaceName,
		catchPointPOUName := __POUNAME(),
		catchPointPosition := __POSITION()
	);

	TryLogDiagnosticException(
		exception := exception,
		severity := TOF_Core.ERROR_SEVERITY.ERROR,
		topic1 := TO_WSTRING(ClassName),
		topic2 := TO_WSTRING(__POUNAME())
	);
__ENDTRY
END_METHOD

(*!
<summary>Invokes reset preparation and converts a callback exception to refusal.</summary>
<description>
Returns TRUE when OnReset returns normally. On exception, formats refuseReason and leaves FALSE. Does not undo
partial reset effects. If obtaining the message raises, retains fixed refusal text. Does not clear terminal
allocation failure; the caller's fatal boundary remains required.
</description>
<param name="refuseReason">Receives formatted diagnostics when reset preparation throws.</param>
*)
METHOD PRIVATE safeCallOnReset : BOOL
VAR_IN_OUT
	refuseReason : TOF_Core.ERROR_MESSAGE;
END_VAR
VAR
	exceptionCode : __SYSTEM.ExceptionCode;	
	exception : TOF_Core.IException;
END_VAR
__TRY
	OnReset();
	
	safeCallOnReset := TRUE;
__CATCH(exceptionCode)
	refuseReason := "Task reset failed";

	__TRY
		exception := TOF_Core.ExceptionManager.GetLastException(
			exceptionCode := exceptionCode,
			catchPointNamespaceName := NamespaceName,
			catchPointPOUName := __POUNAME(),
			catchPointPosition := __POSITION()
		);
		refuseReason := exception.GetMessage();
	__CATCH
		// Keep the fallback text and any terminal allocation-failure latch.
	__ENDTRY
__ENDTRY
END_METHOD

(*!
<summary>Enters READY and clears per-run task state.</summary>
<description>
Used after successful reset preparation. Attempts transition logging, sets StateChanged when the lifecycle
state changes, clears the resource-operation marker, and resets both stop reasons and messages. Does not
release resources or invoke reset hooks.
</description>
*)
METHOD PRIVATE FINAL setIdleState
VAR CONSTANT
	NEW_STATE : TASK_STATE := TASK_STATE.READY;
END_VAR
VAR
	formattedLogMessage : WSTRING(255);
END_VAR
IF _State <> NEW_STATE THEN
	formattedLogMessage := TOF_Core.WideStrings.Concat255(
		"Task '",
		Name,
		"' changed state from '",
		TO_WSTRING(_State),
		"' to '",
		TO_WSTRING(NEW_STATE),
		"'"
	);

	TryLogDiagnosticMessage(
		message := formattedLogMessage,
		category := TOF_Core.LOG_CATEGORY.INFORMATION,
		topic1 := TO_WSTRING(ClassName),
		topic2 := "Task",
		topic3 := TOF_Core.WideStrings.Concat255("Task.", TO_WSTRING(NEW_STATE))
	);

	_State := NEW_STATE;
	_StateChanged := TRUE;
END_IF

_RunningSubstate := TASK_RUNNING_SUBSTATE.PROCESSING;
_ResourceOperationStarted := FALSE;

_OriginalStopReason := TASK_STOP_REASON.WORK_DONE;
_OriginalStopReasonMessage := "";

_FinalStopReason := TASK_STOP_REASON.WORK_DONE;
_FinalStopReasonMessage := "";
END_METHOD

(*!
<summary>Prepares the first execution phase and enters RUNNING.</summary>
<description>
Reads the stable resource manager before publishing RUNNING. Selects acquisition only for a nonzero manager
without an acquired resource, otherwise PROCESSING. Clears stop diagnostics, the resource-operation marker and
the stopping-exception report marker; attempts transition logging. Does not invoke StartAcquire or OnRunning;
Execute advances them.
</description>
*)
METHOD PRIVATE FINAL setRunningState
VAR
	resourceManagerForStart : TOF_Core.IResourceManager;

	formattedLogMessage : WSTRING(255);
END_VAR
VAR CONSTANT
	NEW_STATE : TASK_STATE := TASK_STATE.RUNNING;
END_VAR
resourceManagerForStart := ResourceManager;

IF resourceManagerForStart <> 0 AND_THEN NOT resourceManagerForStart.ResourceAcquired THEN
	setRunningSubstate(runningSubState := TASK_RUNNING_SUBSTATE.RESOURCE_ACQUIRING);
ELSE
	setRunningSubstate(runningSubState := TASK_RUNNING_SUBSTATE.PROCESSING);
END_IF

IF _State <> NEW_STATE THEN
	formattedLogMessage := TOF_Core.WideStrings.Concat255(
		"Task '",
		Name,
		"' changed state from '",
		TO_WSTRING(_State),
		"' to '",
		TO_WSTRING(NEW_STATE),
		"'"
	);

	TryLogDiagnosticMessage(
		message := formattedLogMessage,
		category := TOF_Core.LOG_CATEGORY.INFORMATION,
		topic1 := TO_WSTRING(ClassName),
		topic2 := "Task",
		topic3 := TOF_Core.WideStrings.Concat255("Task.", TO_WSTRING(NEW_STATE))
	);
END_IF

_ResourceOperationStarted := FALSE;
_StoppingExceptionReportAttempted := FALSE;

_OriginalStopReason := TASK_STOP_REASON.WORK_DONE;
_OriginalStopReasonMessage := "";

_FinalStopReason := TASK_STOP_REASON.WORK_DONE;
_FinalStopReasonMessage := "";

IF _State <> NEW_STATE THEN
	_State := NEW_STATE;
	_StateChanged := TRUE;
END_IF
END_METHOD

(*!
<summary>Selects a running phase and resets its one-time resource request marker.</summary>
<description>
Does not format diagnostics, change the lifecycle state or StateChanged, or invoke the resource manager.
</description>
<param name="runningSubState">Phase to execute on the next applicable dispatch.</param>
*)
METHOD PRIVATE setRunningSubstate
VAR_INPUT
	runningSubState : TASK_RUNNING_SUBSTATE;
END_VAR
_RunningSubstate := runningSubState;
_ResourceOperationStarted := FALSE;
END_METHOD

(*!
<summary>Records the final result and enters STOPPED.</summary>
<description>
Attempts transition logging and sets StateChanged on a lifecycle transition. Copies a nonempty supplied
message, otherwise uses the original message or a default for the final reason. Preserves the original reason
and does not itself invoke OnAfterStop. STOPPED does not prove physical resource release.
</description>
<param name="finalStopReason">Final lifecycle result, including any release failure.</param>
<param name="finalStopReasonMessage">
Borrowed diagnostic text copied during this call; may alias the task's original message.
</param>
*)
METHOD PRIVATE FINAL setStoppedState
VAR_INPUT
	finalStopReason : TASK_STOP_REASON;
END_VAR
VAR_IN_OUT CONSTANT
	finalStopReasonMessage : TOF_Core.ERROR_MESSAGE;
END_VAR
VAR CONSTANT
	NEW_STATE : TASK_STATE := TASK_STATE.STOPPED;
END_VAR
VAR
	formattedLogMessage : WSTRING(255);
END_VAR
IF _State <> NEW_STATE THEN
	formattedLogMessage := TOF_Core.WideStrings.Concat255(
		"Task '",
		Name,
		"' changed state from '",
		TO_WSTRING(_State),
		"' to '",
		TO_WSTRING(NEW_STATE),
		"'"
	);

	TryLogDiagnosticMessage(
		message := formattedLogMessage,
		category := TOF_Core.LOG_CATEGORY.INFORMATION,
		topic1 := TO_WSTRING(ClassName),
		topic2 := "Task",
		topic3 := TOF_Core.WideStrings.Concat255("Task.", TO_WSTRING(NEW_STATE))
	);

	_State := NEW_STATE;
	_StateChanged := TRUE;
END_IF

_FinalStopReason := finalStopReason;

IF finalStopReasonMessage <> "" THEN
	_FinalStopReasonMessage := finalStopReasonMessage;
ELSE
	IF _OriginalStopReasonMessage <> "" THEN
		_FinalStopReasonMessage := _OriginalStopReasonMessage;
	ELSE
		CASE _FinalStopReason OF
			TASK_STOP_REASON.WORK_DONE:
				_FinalStopReasonMessage := "Work done";

			TASK_STOP_REASON.INTERNAL_ABORT:
				_FinalStopReasonMessage := "Stopped by internal logic";

			TASK_STOP_REASON.EXTERNAL_CANCEL:
				_FinalStopReasonMessage := "Stopped by external logic";

			TASK_STOP_REASON.FAILURE:
				_FinalStopReasonMessage := "Exception occured";
		END_CASE

	END_IF

END_IF
END_METHOD

(*!
<summary>Starts a prepared task in READY.</summary>
<description>
Returns TRUE after OnBeforeStart succeeds and RUNNING is established; work and acquisition are advanced by
subsequent Execute calls. An ineligible state or a caught preparation failure returns FALSE with refuseReason.
Callback effects are not rolled back. Failure to obtain a callback exception's message uses fixed refusal
text; terminal allocation failure still requires the caller's task-boundary check.
</description>
<param name="refuseReason">Reason for refusal; meaningful when the method returns FALSE.</param>
*)
METHOD FINAL Start : BOOL
VAR_OUTPUT
	refuseReason : TOF_Core.ERROR_MESSAGE;
END_VAR
Start := FALSE;

IF _State <> TASK_STATE.READY THEN
	refuseReason := TOF_Core.WideStrings.Concat255(
		"Expected state is '",
		TO_WSTRING(TASK_STATE.READY),
		"' but current state is '",
		TO_WSTRING(_State),
		"'"
	);
	RETURN;
END_IF

IF safeCallOnBeforeStart(refuseReason := refuseReason) THEN
	setRunningState();

	Start := TRUE;
END_IF
END_METHOD

(*!
<summary>Provides a live read-only lifecycle view.</summary>
<description>
READY permits Start, RUNNING includes work and cleanup, and STOPPED permits result inspection and Reset.
StateChanged is cleared at the beginning of each Execute and set on a lifecycle transition; it is not a global
one-cycle pulse. The view must not outlive this task.
</description>
*)
{attribute 'monitoring' := 'call'}
PROPERTY FINAL State : REFERENCE TO TaskState
GET
State REF= _StateObject;
END_GET
END_PROPERTY

(*!
<summary>Selects a borrowed independent destination for internal task diagnostics.</summary>
<description>
Zero uses the existing LogManager filtering, numbering and routing. A nonzero destination is called directly,
without LogManager or its filter/counters, and must not return to the active logging chain. Configure before
Start and keep it stable and alive through STOPPED and Reset. The task does not own, configure or execute
the destination. Assignment performs no I/O or callbacks; one owner task provides synchronization.
</description>
*)
PROPERTY FINAL DiagnosticLogger : TOF_Core.ILogger
GET
DiagnosticLogger := _DiagnosticLogger;
END_GET
SET
_DiagnosticLogger := DiagnosticLogger;
END_SET
END_PROPERTY

(*!
<summary>Reports an internal message through the configured diagnostic route.</summary>
<description>
Uses the borrowed DiagnosticLogger directly when present; otherwise retains LogManager topics and routing.
Contains destination exceptions without recursive logging. Returns FALSE on observed terminal allocation
failure; prior diagnostic effects are not rolled back and the fatal latch remains set.
</description>
*)
METHOD PROTECTED FINAL TryLogDiagnosticMessage : BOOL
VAR_IN_OUT CONSTANT
	message : TOF_Core.ERROR_MESSAGE;
END_VAR
VAR_INPUT
	category : TOF_Core.LOG_CATEGORY;
	topic1 : WSTRING := "";
	topic2 : WSTRING := "";
	topic3 : WSTRING := "";
END_VAR
__TRY

	IF TOF_Core.DynamicMemoryManager.HasAllocationFailed THEN
		RETURN;
	END_IF

	IF _DiagnosticLogger <> 0 THEN
		TryLogDiagnosticMessage := _DiagnosticLogger.TryLogMessage(category := category, message := message);
	ELSE
		TryLogDiagnosticMessage := TOF_Core.LogManager.TryLogMessage(
			category := category,
			message := message,
			topic1 := topic1,
			topic2 := topic2,
			topic3 := topic3
		);
	END_IF

	IF TOF_Core.DynamicMemoryManager.HasAllocationFailed THEN
		TryLogDiagnosticMessage := FALSE;
	END_IF

__CATCH
	// Diagnostic failure must not replace the task lifecycle outcome.
	TryLogDiagnosticMessage := FALSE;
__ENDTRY
END_METHOD

(*!
<summary>Reports an internal exception through the configured diagnostic route.</summary>
<description>
Uses the borrowed DiagnosticLogger directly when present; otherwise retains LogManager topics and routing.
Contains destination exceptions without recursive logging. Returns FALSE on observed terminal allocation
failure; prior diagnostic effects are not rolled back and the fatal latch remains set.
</description>
*)
METHOD PROTECTED FINAL TryLogDiagnosticException : BOOL
VAR_INPUT
	exception : TOF_Core.IReadOnlyException;
	severity : TOF_Core.ERROR_SEVERITY;
	topic1 : WSTRING := "";
	topic2 : WSTRING := "";
	topic3 : WSTRING := "";
END_VAR
__TRY

	IF TOF_Core.DynamicMemoryManager.HasAllocationFailed THEN
		RETURN;
	END_IF

	IF _DiagnosticLogger <> 0 THEN
		TryLogDiagnosticException := _DiagnosticLogger.TryLogException(exception := exception, severity := severity);
	ELSE
		TryLogDiagnosticException := TOF_Core.LogManager.TryLogException(
			exception := exception,
			severity := severity,
			topic1 := topic1,
			topic2 := topic2,
			topic3 := topic3
		);
	END_IF

	IF TOF_Core.DynamicMemoryManager.HasAllocationFailed THEN
		TryLogDiagnosticException := FALSE;
	END_IF

__CATCH
	// Diagnostic failure must not replace the task lifecycle outcome.
	TryLogDiagnosticException := FALSE;
__ENDTRY
END_METHOD

END_FUNCTION_BLOCK

// ---- Task/SubObjects/TaskState.TcPOU
(*
SPDX-FileCopyrightText: Â© 2026 Oleksandr Tiutyk <trofimich@gmail.com>
SPDX-License-Identifier: MIT
License: https://opensource.org/license/mit
*)

(*!
<summary>Exposes the task lifecycle and transition indicator for observation.</summary>
<description>
Borrows live backing variables supplied at initialization or rebound after online change. Getters safely guard
against unbound references and return default values if references are not valid. Treat the view and returned
references as read-only. Copy values when a snapshot is required.
</description>
*)

FUNCTION_BLOCK FINAL TaskState
VAR
	{attribute 'hide'} 
	_TaskState : REFERENCE TO TASK_STATE;
	{attribute 'hide'} 
	_TaskStateChanged : REFERENCE TO BOOL;
END_VAR

(*!
<summary>Binds the view to its owner's live state.</summary>
<description>
Stores references without copying their current values or changing the owner. Valid supplied references are
bound; skipped during online change copy code. Does not allocate or raise framework exceptions.
</description>
<param name="taskState">Live lifecycle state owned by the task.</param>
<param name="taskStateChanged">Live transition indicator owned by the task.</param>
*)
METHOD FB_Init: BOOL
VAR_INPUT
	bInitRetains : BOOL; // TRUE: the retain variables are initialized (reset warm / reset cold)
	bInCopyCode : BOOL;  // TRUE: the instance will be copied to the copy code afterward (online change)
	taskState : REFERENCE TO TASK_STATE;
	taskStateChanged : REFERENCE TO BOOL;
END_VAR
IF NOT bInCopyCode THEN
	Rebind(
		taskState := taskState,
		taskStateChanged := taskStateChanged
	);
END_IF
END_METHOD

(*!
<summary>Reports whether the task is READY.</summary>
<description>
READY permits Start; it does not imply a completed previous run. Returns FALSE if unbound.
</description>
*)
{attribute 'monitoring' := 'call'}
PROPERTY FINAL Ready : BOOL
GET
IF __ISVALIDREF(_TaskState) THEN
	Ready := _TaskState = TASK_STATE.READY;
END_IF
END_GET
END_PROPERTY

(*!
<summary>Rebinds the view to its owner's live state variables.</summary>
<description>
Updates internal references when valid variables are supplied. Used during initialization and
subsequent online-change reinitialization.
</description>
<param name="taskState">Live lifecycle state owned by the task.</param>
<param name="taskStateChanged">Live transition indicator owned by the task.</param>
*)
METHOD INTERNAL Rebind
VAR_INPUT
	taskState : REFERENCE TO TASK_STATE;
	taskStateChanged : REFERENCE TO BOOL;
END_VAR
IF __ISVALIDREF(taskState) THEN
	_TaskState REF= taskState;
END_IF

IF __ISVALIDREF(taskStateChanged) THEN
	_TaskStateChanged REF= taskStateChanged;
END_IF
END_METHOD

(*!
<summary>Reports whether the task is RUNNING.</summary>
<description>
Includes acquisition, processing, stopping and resource release. Returns FALSE if unbound.
</description>
*)
{attribute 'monitoring' := 'call'}
PROPERTY FINAL Running : BOOL
GET
IF __ISVALIDREF(_TaskState) THEN
	Running := _TaskState = TASK_STATE.RUNNING;
END_IF
END_GET
END_PROPERTY

(*!
<summary>Reports a lifecycle transition since the last Execute began.</summary>
<description>
Task.Execute clears this flag on entry, including when not running. Start, stopping and successful reset from
STOPPED can set it. It is not a count or a pulse tied to all PLC cycles. Returns FALSE if unbound.
</description>
*)
{attribute 'monitoring' := 'call'}
PROPERTY FINAL StateChanged : BOOL
GET
IF __ISVALIDREF(_TaskStateChanged) THEN
	StateChanged := _TaskStateChanged;
END_IF
END_GET
END_PROPERTY

(*!
<summary>Reports whether the task is STOPPED.</summary>
<description>
Read FinalStopReason for the result; stopping does not prove physical release. Returns FALSE if unbound.
</description>
*)
{attribute 'monitoring' := 'call'}
PROPERTY FINAL Stopped : BOOL
GET
IF __ISVALIDREF(_TaskState) THEN
	Stopped := _TaskState = TASK_STATE.STOPPED;
END_IF
END_GET
END_PROPERTY

(*!
<summary>Returns the current lifecycle state by value.</summary>
<description>
The returned enum is a snapshot of the borrowed backing state at this read. Returns READY if unbound.
</description>
*)
{attribute 'monitoring' := 'call'}
PROPERTY FINAL Value : TASK_STATE
GET
IF __ISVALIDREF(_TaskState) THEN
	Value := _TaskState;
END_IF
END_GET
END_PROPERTY

END_FUNCTION_BLOCK
